FUNCTION_BLOCK P_Choice (* Exclusive gateway: EO_TRUE if the Cond parameter is TRUE, else EO_FALSE *)
  (* Standard: 61499-2 *)
  (* Version 2.0, 2026-09-27, Project contributors, Filling cell reference model *)
  PACKAGE fillingcell;
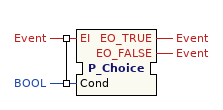
  EVENT_INPUT
    EI WITH Cond;
  END_EVENT
  EVENT_OUTPUT
    EO_TRUE;
    EO_FALSE;
  END_EVENT
  VAR_INPUT
    Cond : BOOL;
  END_VAR
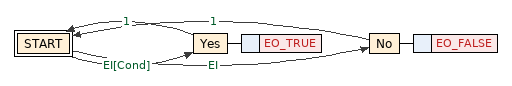
  EC_STATES
    START;
    Yes : -> EO_TRUE;
    No : -> EO_FALSE;
  END_STATES
  EC_TRANSITIONS
    START TO Yes := EI[Cond];
    START TO No := EI;
    Yes TO START := 1;
    No TO START := 1;
  END_TRANSITIONS
END_FUNCTION_BLOCK
